PROGRAM MAIN

VAR CONSTANT
	SAMPLE_SIZE : INT := 1000;
END_VAR

VAR_INPUT
	logActive : BOOL := FALSE;
	MTSendString : STRING(132) := 'SIR$0D$0A';
	//Pump control
	P9999A : sMasterflexPort := (bDirection := FALSE, nTubeSize := 13);
	P9999B : sMasterflexPort := (bDirection := FALSE, nTubeSize := 16);
	//totalizer blocks
	fbFQ9999A : FQ1;
	fbFQ9999B : FQ1;
	fbFQ9999C : FQ1;
	
	phase : UINT := 0;
	//Flow and Concentration Control
	FC9999A1 : FC1;
	FC9999A2 : FC1b;
	FC9999B1 : FC1;
	FC9999B2 : FC1b;
	FCForm : UINT := 2;
	AC9999C : CC1;
	FV9999C : FV3;
	FVC9999C : FVC3;

END_VAR

VAR
	//test
    Tau : LREAL := 1.0;
	FilterFactor : LREAL;
	ftfirstorder : LREAL;
	//-test
	heartbeat : DINT;
	fbGetUnixTimeGlobal : fbGetUnixTime;
	temp : UINT;
	MTWeight : sWeight;
	
	//Flowmeters
	FT9999A : AI := (loCutEnable:= FALSE, loCut := 0.25, scale := (euLo := -20.0,  euHi := 100.0, eu := 'ml/min')); //E+H small
	FT9999B : AI := (loCutEnable:= TRUE, loCut := 2.25, scale := (euLo := 0,  euHi := 1000.0, eu := 'ml/min')); //E+H large
	FT9999C : AI := (loCutEnable:= TRUE, loCut := 2.25, scale := (euLo := 0,  euHi := 1000.0, eu := 'ml/min')); //E+H very large
	
	//Pressures
	PT9999A : AI := (scale := (euLo := 0,  euHi := 15.0, eu := 'psig'));
	PT9999B : AI := (scale := (euLo := 0,  euHi := 15.0, eu := 'psig'));
	PT9999C : AI := (scale := (euLo := 0,  euHi := 15.0, eu := 'psig'));

	//Reveal
	AT9999RV290 : AI := (scale := (euLo := -0.1,  euHi := 2.0, eu := 'AU'));
	AT9999RV300 : AI := (scale := (euLo := -0.1,  euHi := 1.1, eu := 'mg/ml'));
	AT9999RV310 : AI := (scale := (euLo := 0,  euHi := 2.0, eu := 'AU'));
	AT9999RV320 : AI := (scale := (euLo := 0,  euHi := 2.0, eu := 'AU'));
	AT9999C : ModbusTCPReveal();

	//ColorWise
	AT9999CWx  : AI := (scale := (rawLo := 0, rawHi := 16383, euLo := 0,  euHi := 1.0, eu := 'x'));
	AT9999CWy  : AI := (scale := (rawLo := 0, rawHi := 16383, euLo := 0,  euHi := 1.0, eu := 'y'));
	AT9999CWYY : AI := (scale := (rawLo := 0, rawHi := 16383, euLo := 0,  euHi := 1.0, eu := 'Y'));

	//function blocks
	fbP9999A : fbMasterflex;
	fbP9999B : fbMasterflex;
	
	//Phases
	FT9999A_FLOWCAL : FlowCalSequence;
	FT9999B_FLOWCAL : FlowCalSequence;
	
	//AI blocks
	fbFT9999A : AI1;
	fbFT9999B : AI1;
	fbFT9999C : AI1;
	fbPT9999A : AI1;
	fbPT9999B : AI1;
	fbPT9999C : AI1;
	fbAT9999RV290 : AI1;
	fbAT9999RV300 : AI1;
	fbAT9999RV310 : AI1;
	fbAT9999RV320 : AI1;
	fbAT9999CWx  : AI1;
	fbAT9999CWy  : AI1;
	fbAT9999CWYY : AI1;
	
	// filter blocks
	fbFT9999AFilt : fbMovingAverage;
	FT9999ASize : UINT := 500;
	FT9999AFiltTarget : LREAL := 1500.0; //Target number of ms to for moving average
	fbFT9999BFilt : fbMovingAverage;
	FT9999BSize : UINT := 500;
	FT9999BFiltTarget : LREAL := 1500.0; //Target number of ms to for moving average
	fbFT9999CFilt : fbMovingAverage;
	FT9999CSize : UINT := 500;
	fbFT9999CfqFilt : fbMovingAverage;

	//Data logging
	fbP9999ARPMlog : fbDatalogger_100ms;
	fbP9999AFlowlog : fbDatalogger_100ms;
	fbP9999BRPMlog : fbDatalogger_100ms;
	fbP9999BFlowlog : fbDatalogger_100ms;
		
	fbFT9999Alog : fbDatalogger_1ms;
	fbFT9999Blog : fbDatalogger_1ms;
	fbFT9999Clog : fbDatalogger_1ms;
	
	fbFT9999Afiltlog : fbDatalogger_100ms;
	fbFT9999Bfiltlog : fbDatalogger_100ms;
	fbFT9999Cfiltlog : fbDatalogger_100ms;
	
	fbFQ9999Alog : fbDatalogger_100ms;
	fbFQ9999Blog : fbDatalogger_100ms;
	fbFQ9999Clog : fbDatalogger_100ms;
	
	fbPT9999Alog : fbDatalogger_1ms;
	fbPT9999Blog : fbDatalogger_1ms;
	fbPT9999Clog : fbDatalogger_1ms;

	fbWT9999Clog : fbDatalogger_100ms;

	fbAT9999RV290log : fbDatalogger_10ms;
	fbAT9999RV300log : fbDatalogger_10ms;
	fbAT9999RV310log : fbDatalogger_10ms;
	fbAT9999RV320log : fbDatalogger_10ms;

	fbAT9999CWxlog  : fbDatalogger_1ms;
	fbAT9999CWylog  : fbDatalogger_1ms;
	fbAT9999CWYYlog : fbDatalogger_1ms;
	
END_VAR

heartbeat := heartbeat + 1;
fbGetUnixTimeGlobal();  //set global variable unixTime
//Code that runs 1 time per second
IF (heartbeat MOD 1000) = 0 THEN
	temp := MIN(2499,DINT_TO_UINT(3*TRUNC(P9999A.fPeriodMS)));  //lower bound is 3 * period - want to make sure at least 3 periods are averaged
	FT9999ASize := LIMIT(temp, DINT_TO_UINT((TRUNC(P9999A.fPeriodMS) * TRUNC(FT9999AFiltTarget/P9999A.fPeriodMS))), 2500);
	temp := MIN(2499,DINT_TO_UINT(3*TRUNC(P9999B.fPeriodMS)));  //lower bound is 3 * period - want to make sure at least 3 periods are averaged
	FT9999BSize := LIMIT(temp, DINT_TO_UINT((TRUNC(P9999B.fPeriodMS) * TRUNC(FT9999BFiltTarget/P9999B.fPeriodMS))), 2500);
END_IF

//Call serial line handlers
MTSerial(sSendString := MTSendString, weight := MTWeight);

//Call pump handler
fbP9999A(sPort := P9999A);
fbP9999B(sPort := P9999B);

//Valve handlers
fv9999c();


//Flow transmitters
fbFT9999A(AI := FT9999A);
fbFT9999AFilt(in := FT9999A.pv, size := FT9999ASize, out => FT9999A.pvfilt);

//test
FilterFactor := 1.0 - EXP(-0.001/tau);
ftfirstorder := (1.0 - filterfactor) * ftfirstorder + filterfactor * FT9999A.pv;
//-test


fbFQ9999A(flow := FT9999A.pv, timeBaseMS := (1000.0*60.0));
fbFT9999B(AI := FT9999B);
fbFT9999BFilt(in := FT9999B.pv, size := FT9999BSize, out => FT9999B.pvfilt);
fbFQ9999B(flow := FT9999B.pv, timeBaseMS := (1000.0*60.0));
fbFT9999C(AI := FT9999C);
fbFT9999CFilt(in := FT9999C.pv, size := FT9999CSize, out => FT9999C.pvfilt);
fbFQ9999C(flow := FT9999C.pv, timeBaseMS := (1000.0*60.0));

//Flow and Concentration Control
IF FCForm = 1 THEN
	FC9999A1(FTOLS := FT9999A_OLS, pumpOLS := P9999A_OLS, pump := P9999A, ft := FT9999A, sPID := FC9999A1CtrlData);
	FC9999B1(FTOLS := FT9999B_OLS, pumpOLS := P9999B_OLS, pump := P9999B, ft := FT9999B, sPID := FC9999B1CtrlData);
ELSIF FCForm = 2 THEN
	FC9999A2(FTOLS := FT9999A_OLS, pumpOLS := P9999A_OLS, pump := P9999A, ft := FT9999A, ctrlData:= FC9999ACtrlData);
	FC9999B2(FTOLS := FT9999B_OLS, pumpOLS := P9999B_OLS, pump := P9999B, ft := FT9999B, ctrlData:= FC9999BCtrlData);
END_IF
FT9999A_FLOWCAL(fq := fbFQ9999A, pump := P9999A, FTOLS := FT9999A_OLS, pumpOLS := P9999A_OLS);
FT9999B_FLOWCAL(fq := fbFQ9999B, pump := P9999B, FTOLS := FT9999B_OLS, pumpOLS := P9999B_OLS);
AC9999C(FCA := FC9999A2, FTA := FT9999A, FCB:= FC9999B2, FTB := FT9999B, PumpA := P9999A, PumpB := P9999B);
//FVC9999C(conc := AT9999C.pv, FTA := FT9999A, FTB := FT9999B, FV := FV9999C, PumpA := P9999A, PumpB := P9999B, FTC := AT9999C);

//Pressure
fbPT9999A(AI := PT9999A);
fbPT9999B(AI := PT9999B);
fbPT9999C(AI := PT9999C);

//Reveal
fbAT9999RV290(AI := AT9999RV290);
fbAT9999RV300(AI := AT9999RV300);
fbAT9999RV310(AI := AT9999RV310);
fbAT9999RV320(AI := AT9999RV320);
AT9999C();

//ColorWise
fbAT9999CWx(AI := AT9999CWx);
fbAT9999CWy(AI := AT9999CWy);
fbAT9999CWYY(AI := AT9999CWYY);

//Data Logging
fbP9999ARPMlog(fData := P9999A.fSpeedPV);
fbP9999AFlowlog(fData := P9999A.fFlowPV);
fbP9999BRPMlog(fData := P9999B.fSpeedPV);
fbP9999BFlowlog(fData := P9999B.fFlowPV);
	
fbFT9999Alog(fData := FT9999A.pv);;
fbFT9999Blog(fData := FT9999B.pv);
fbFT9999Clog(fData := FT9999C.pv);

fbFT9999Afiltlog(fData := FT9999A.pvfilt);
fbFT9999Bfiltlog(fData := FT9999B.pvfilt);
fbFT9999Cfiltlog(fData := FT9999C.pvfilt);

fbFQ9999Alog(fData := fbFQ9999A.total);
fbFQ9999Blog(fData := fbFQ9999B.total);
fbFQ9999Clog(fData := fbFQ9999C.total);

fbPT9999Alog(fData := PT9999A.pv);
fbPT9999Blog(fData := PT9999B.pv);
fbPT9999Clog(fData := PT9999C.pv);

fbWT9999Clog(fData := MTWeight.pv);

fbAT9999RV290log(fData := AT9999RV290.pv);
fbAT9999RV300log(fData := AT9999RV300.pv);
fbAT9999RV310log(fData := AT9999RV310.pv);
fbAT9999RV320log(fData := AT9999RV320.pv);

fbAT9999CWxlog(fData := AT9999CWx.pv);
fbAT9999CWylog(fData := AT9999CWy.pv);
fbAT9999CWYYlog(fData := AT9999CWYY.pv);

//Phase Control
CASE phase OF
1:
	FT9999A_FLOWCAL.start := TRUE;
	phase := 0;
2:
	FT9999B_FLOWCAL.start := TRUE;
	phase := 0;
END_CASE

END_PROGRAM

(* stored: Version 1.1.0.1, ProductVersion 3.1.0.36
   POU MAIN: Id {ef40301a-07cc-419a-94a7-572c9743ae72}, SpecialFunc None *)
